PROGRAM PRG_1_PlcTask
VAR
END_VAR

PRG_MR1K4_SOMS();
PRG_MR2K4_KBO();
PRG_MR3K4_KBO();
PRG_MR4K4_KBO();
PRG_MR5K4_KBO();

END_PROGRAM

(* stored: Version 1.1.0.1, ProductVersion 3.1.4024.12
   POU PRG_1_PlcTask: Id {3f92f9bc-a1dd-43f7-bd6e-fa51ae4184b4}, SpecialFunc None *)
